// TIA Portal V16 export
// export: Created 2026-06-18T03:48:04.5137603Z, ExportSetting WithDefaults, DisplayName Totally Integrated Automation Portal, DisplayVersion V16 Update 8, DisplayName TIA Portal Version Control Interface, DisplayVersion V16 Update 8, DisplayName TIA Portal Openness, DisplayVersion V16 Update 8, DisplayName SINAMICS Startdrive Advanced, DisplayVersion V16, DisplayName SINAMICS Startdrive G130, G150, S120, S150, SINAMICS MV, S210, DisplayVersion V16, DisplayName SINAMICS Startdrive G110M, G120, G120C, G120D, G120P, DisplayVersion V16, DisplayName STEP 7 Professional, DisplayVersion V16 Update 8, DisplayName STEP 7 Safety, DisplayVersion V16 Update 7, DisplayName WinCC Advanced, DisplayVersion V16 Update 8
Screen "Login_Screen"  1280x800, Number=1
  ScreenLayer 
    IOField "IO_Password" at 460,260 size 240x44  DataFormat=Decimal, FormatPattern=9999999, Mode=InOutput
    Button "BTN_Logout" at 590,360 size 110x50  Mode=Text, HelpText="退出", TextOff="Text", TextOn="Text"
    SymbolicIOField "符号 I/O 域_1" at 177,87 size 170x32  CountVisibleItems=3, Mode=InOutput, OnValue=1, TextOff="0", TextOn="1"
    Circle "LMP_Online" at 840,270 size 48x48
    TextField "TXT_Title" at 440,60 size 400x48  Text="操作员登录Text"
